FUNCTION_BLOCK FB_ReadTechnoGFunc
VAR_INPUT
   sNetId               : T_AmsNetId;
   nPort                : T_AmsPort := 553;
   nIdxGrp              : UDINT;
   nIdxOffs             : UDINT;
	nLen						: UDINT;
   bStart               : BOOL;
	pStr						: POINTER TO STRING;
END_VAR
VAR_OUTPUT
   bBusy                : BOOL;
   bErr                 : BOOL;
END_VAR
VAR
   fbRead               : ADSREAD;
   bStarted             : BOOL;
   destArr               : ARRAY[0..40] OF INT;
	i							: INT;
	tmp						: STRING;
END_VAR

(* ========================================================= *)
(*     FB: FB_ReadTechnoGFunc                                *)
(* --------------------------------------------------------- *)
(*   Desc: Reads the technology information                  *)
(*       : from the CNC                                      *)
(* Author: MK                                                *)
(*   Date: 21.12.2011                                        *)
(*   Rev.: 1.0                                               *)
(* ========================================================= *)


IF bStart = TRUE AND bStarted = FALSE THEN
	bStarted := TRUE;
	bErr := FALSE;
	bBusy := TRUE;
END_IF

IF bStarted THEN
   fbRead(NetID:=sNetId, Port:=nPort, IdxGrp:=nIdxGrp, IdxOffs:=nIdxOffs,
         LEN:=nLen, DestAddr:=ADR(destArr), READ:=bStarted, TMOUT:=DEFAULT_ADS_TIMEOUT);
   IF NOT fbRead.Busy THEN
      IF fbRead.Err THEN
         bErr := TRUE;
		ELSE
			tmp := '';
			FOR i:=0 TO 36 DO
				IF destArr[i] <> -1 THEN
					tmp := CONCAT(tmp, 'G');
					tmp := CONCAT(tmp, INT_TO_STRING(destArr[i]));
					tmp := CONCAT(tmp, ' ');
		      END_IF
			END_FOR
			pStr^ := tmp;
      END_IF
      fbRead(READ := FALSE);
      bStarted := FALSE;
      bBusy := FALSE;
   END_IF
END_IF

END_FUNCTION_BLOCK

(* stored: Version 1.1.0.1, ProductVersion 3.1.4020.6
   POU FB_ReadTechnoGFunc: Id {4b1393c8-523c-410e-b09c-45befccef323}, SpecialFunc None *)
